INTERFACE I_AsynchronousRpcResponse EXTENDS I_Disposable

METHOD PUBLIC CompleteWithBase64
VAR_INPUT
	pBytes : POINTER TO BYTE;
	nBytes : DINT;
END_VAR
END_METHOD

METHOD PUBLIC CompleteWithBool
VAR_INPUT
	Value : BOOL;
END_VAR
END_METHOD

METHOD PUBLIC CompleteWithBytesAsHex
VAR_INPUT
	pBytes : POINTER TO BYTE;
	nBytes : DINT;
END_VAR
END_METHOD

METHOD PUBLIC CompleteWithDateTime
VAR_INPUT
	Value : DATE_AND_TIME;
END_VAR
END_METHOD

METHOD PUBLIC CompleteWithDcTime
VAR_INPUT
	Value : DCTIME;
END_VAR
END_METHOD

METHOD PUBLIC CompleteWithDint
VAR_INPUT
	Value : DINT;
END_VAR
END_METHOD

METHOD PUBLIC CompleteWithFileTime
VAR_INPUT
	Value : FILETIME;
END_VAR
END_METHOD

METHOD PUBLIC CompleteWithLint
VAR_INPUT
	Value : LINT;
END_VAR
END_METHOD

METHOD PUBLIC CompleteWithLreal
VAR_INPUT
	Value : LREAL;
END_VAR
END_METHOD

METHOD PUBLIC CompleteWithNull
VAR_INPUT
END_VAR
END_METHOD

METHOD PUBLIC CompleteWithObject
VAR_INPUT
	Object : I_Serializable;
END_VAR
END_METHOD

METHOD PUBLIC CompleteWithReal
VAR_INPUT
	Value : REAL;
END_VAR
END_METHOD

METHOD PUBLIC CompleteWithSerializer
VAR_INPUT
	Serializer : I_Serializer;
END_VAR
END_METHOD

METHOD PUBLIC CompleteWithString
VAR_INPUT
	Value : T_MAXSTRING;
END_VAR
END_METHOD

METHOD PUBLIC CompleteWithUdint
VAR_INPUT
	Value : UDINT;
END_VAR
END_METHOD

METHOD PUBLIC CompleteWithUlint
VAR_INPUT
	Value : ULINT;
END_VAR
END_METHOD

METHOD PUBLIC GetSerializer : I_Serializer
VAR_INPUT
END_VAR
END_METHOD

METHOD PUBLIC RejectWithMessage
VAR_INPUT
	Message : T_MAXSTRING;
END_VAR
END_METHOD

END_INTERFACE

(* stored: Version 1.1.0.1, ProductVersion 3.1.4024.12
   Itf I_AsynchronousRpcResponse: Id {654145e2-0cc3-4690-8619-88bc8eafb112}
   Method CompleteWithBase64: Id {432e1430-be65-4e79-8947-57d45859375f}
   Method CompleteWithBool: Id {d4e5ec1e-4234-4825-9f6f-6cb0a5396ae7}
   Method CompleteWithBytesAsHex: Id {5bc8327e-1c3b-4682-87f8-cb6745dd2ab1}
   Method CompleteWithDateTime: Id {f3cb6198-b749-4f4b-8f4c-d8a0c4ab4540}
   Method CompleteWithDcTime: Id {24ba6c53-5e38-4685-a4db-7c7b4612637e}
   Method CompleteWithDint: Id {05dff308-f0b3-4a70-a76d-5da2f3c1aad7}
   Method CompleteWithFileTime: Id {9e04f4ad-1387-4753-a283-49bf87c003b1}
   Method CompleteWithLint: Id {e33d460b-b43f-4181-8cf5-46f81bb60ae5}
   Method CompleteWithLreal: Id {82954cc7-a75d-4ee6-ac2a-6d6cd8cf94fc}
   Method CompleteWithNull: Id {83c10e38-1d12-4a99-8469-a0ea30c17bd1}
   Method CompleteWithObject: Id {080511d1-0593-4fbb-85ac-40064431e848}
   Method CompleteWithReal: Id {26953f8c-4d08-4ef7-ad61-487977a89bd1}
   Method CompleteWithSerializer: Id {70bba3bc-507f-415e-931e-9633d1b43a6a}
   Method CompleteWithString: Id {8330278c-45da-42b8-b740-e05615cb66ce}
   Method CompleteWithUdint: Id {c1a8e854-abb0-4b9d-9af2-71f98e9a8d0d}
   Method CompleteWithUlint: Id {d088e789-5ae8-4618-a498-de9b68f32600}
   Method GetSerializer: Id {2b6e2995-f990-4c69-bab2-54a4ad1a601d}
   Method RejectWithMessage: Id {a3f564bc-c6e0-45b8-bc41-586ee0918ab2} *)
